// TIA Portal V19 export
TYPE "typeSyncNode"
TITLE = typeEquipmentC_SyncNode
// Module synchronous control nodes including synchronous control nodes from child modules
// stored: Namespace Unit.Em2
   STRUCT
      commands { ExternalWritable := 'False'} : Struct   // Example of commands. Must be adjusted depending on the application.
         enableHpMotion : Bool;   // Enable High performance motion program
      END_STRUCT;
      status { ExternalWritable := 'False'} : Struct   // Example of status bits. Must be adjusted depending on the application.
         busy : Bool;   // Logic that is executed in the motion cycle is busy
         error : Bool;   // Logic that is executed in the motion cycle has an error
      END_STRUCT;
   END_STRUCT;
END_TYPE
